% RSLogix 500 project TRAFFIC LIGHT.RSS, saved by version 8.30.00.16 %
PROJECT "UNTITLED"    % processor: MicroLogix 1000 %

PROGRAM FILES
  LAD 2 "MAIN_PROG"  11 rungs
  LAD 3 "FLASHER"  5 rungs
  LAD 4 "TIMER"  8 rungs
  LAD 5 "STI_INT"  1 rungs
  LAD 6, 7, 8, 9, 10, 11, 12, 13, 14, 15, 16: only END

DATA FILES
  O0 OUTPUT  1 elements
  I1 INPUT  2 elements
  S2 STATUS  33 elements
  B3 BINARY  32 elements
  T4 TIMER  40 elements
  C5 COUNTER  32 elements
  R6 CONTROL  16 elements
  N7 INTEGER  105 elements

LADDER 2 "MAIN_PROG"
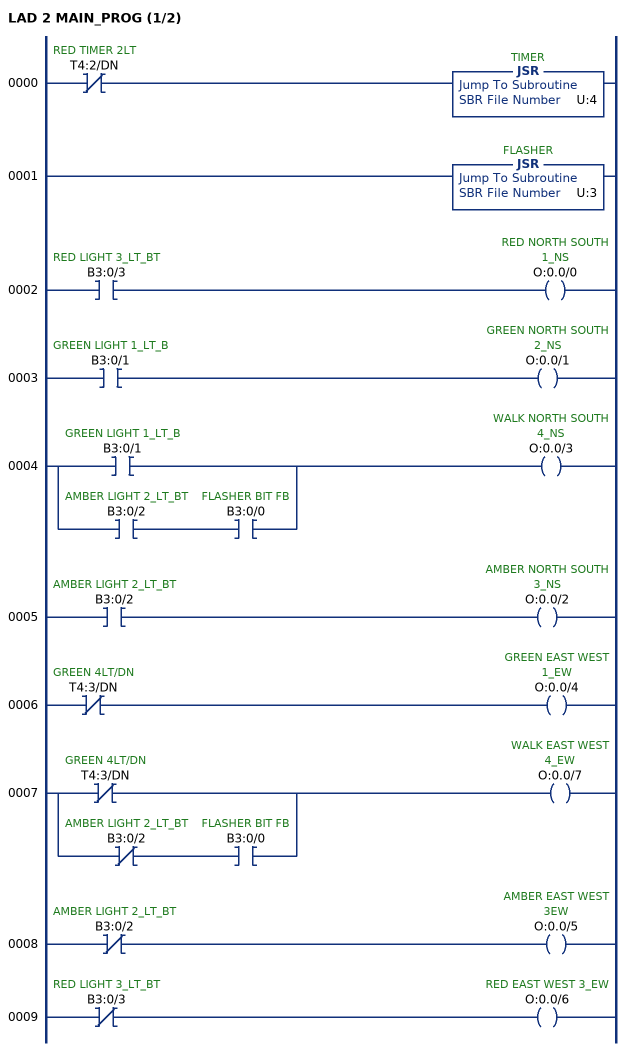
% Rung: 0 %
SOR XIO T4:2/DN JSR U:4 EOR
%   T4:2/DN  2LT  "RED TIMER" %
%   U:4  "TIMER" %
% Rung: 1 %
SOR JSR U:3 EOR
%   U:3  "FLASHER" %
% Rung: 2 %
SOR XIC B3:0/3 OTE O:0.0/0 EOR
%   B3:0/3  3_LT_BT  "RED LIGHT" %
%   O:0.0/0  1_NS  "RED NORTH SOUTH" %
% Rung: 3 %
SOR XIC B3:0/1 OTE O:0.0/1 EOR
%   B3:0/1  1_LT_B  "GREEN LIGHT" %
%   O:0.0/1  2_NS  "GREEN NORTH SOUTH" %
% Rung: 4 %
SOR BST XIC B3:0/1 NXB XIC B3:0/2 XIC B3:0/0 BND OTE O:0.0/3 EOR
%   B3:0/1  1_LT_B  "GREEN LIGHT" %
%   B3:0/2  2_LT_BT  "AMBER LIGHT" %
%   B3:0/0  FB  "FLASHER BIT" %
%   O:0.0/3  4_NS  "WALK NORTH SOUTH" %
% Rung: 5 %
SOR XIC B3:0/2 OTE O:0.0/2 EOR
%   B3:0/2  2_LT_BT  "AMBER LIGHT" %
%   O:0.0/2  3_NS  "AMBER NORTH SOUTH" %
% Rung: 6 %
SOR XIO T4:3/DN OTE O:0.0/4 EOR
%   T4:3  4LT  "GREEN" %
%   O:0.0/4  1_EW  "GREEN EAST WEST" %
% Rung: 7 %
SOR BST XIO T4:3/DN NXB XIO B3:0/2 XIC B3:0/0 BND OTE O:0.0/7 EOR
%   T4:3  4LT  "GREEN" %
%   B3:0/2  2_LT_BT  "AMBER LIGHT" %
%   B3:0/0  FB  "FLASHER BIT" %
%   O:0.0/7  4_EW  "WALK EAST WEST" %
% Rung: 8 %
SOR XIO B3:0/2 OTE O:0.0/5 EOR
%   B3:0/2  2_LT_BT  "AMBER LIGHT" %
%   O:0.0/5  3EW  "AMBER EAST WEST" %
% Rung: 9 %
SOR XIO B3:0/3 OTE O:0.0/6 EOR
%   B3:0/3  3_LT_BT  "RED LIGHT" %
%   O:0.0/6  3_EW  "RED EAST WEST" %

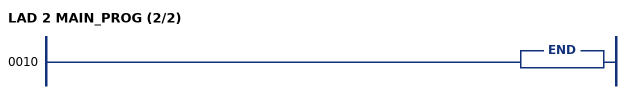
% Rung: 10 %
SOR END EOR

LADDER 3 "FLASHER"
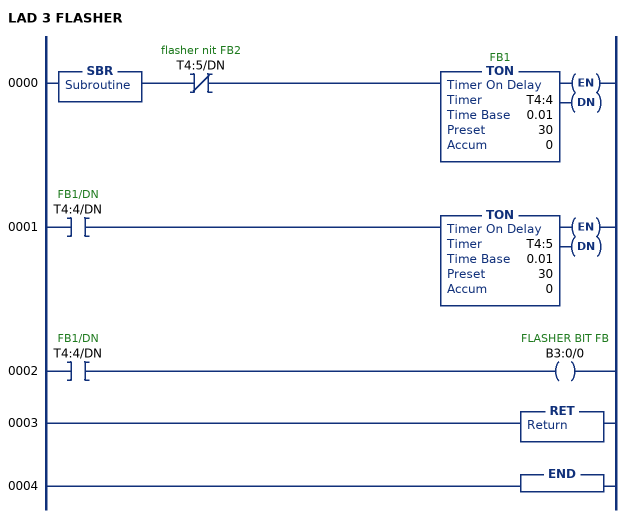
% Rung: 0 %
SOR SBR XIO T4:5/DN TON T4:4 0.01 30 0 EOR
%   T4:5/DN  FB2  "flasher nit" %
%   T4:4  FB1 %
% Rung: 1 %
SOR XIC T4:4/DN TON T4:5 0.01 30 0 EOR
%   T4:4  FB1 %
% Rung: 2 %
SOR XIC T4:4/DN OTE B3:0/0 EOR
%   T4:4  FB1 %
%   B3:0/0  FB  "FLASHER BIT" %
% Rung: 3 %
SOR RET EOR
% Rung: 4 %
SOR END EOR

LADDER 4 "TIMER"
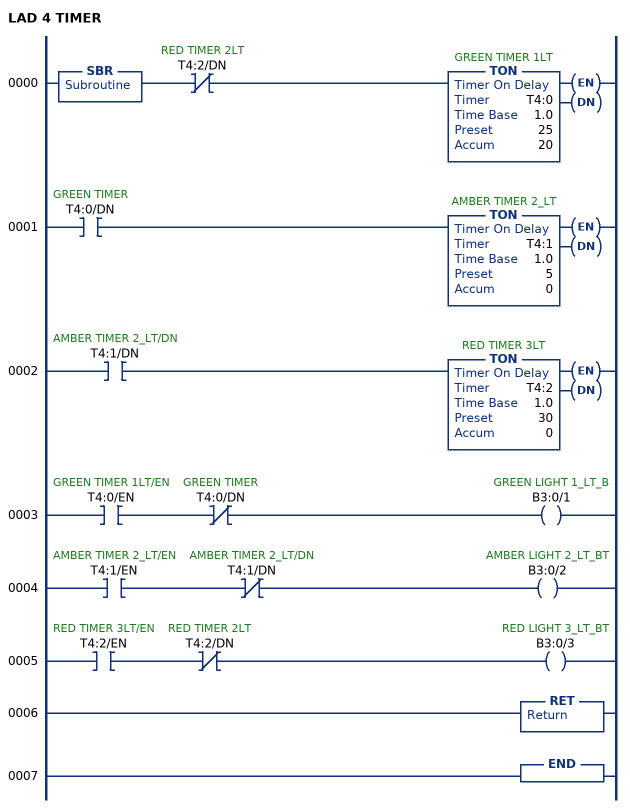
% Rung: 0 %
SOR SBR XIO T4:2/DN TON T4:0 1.0 25 20 EOR
%   T4:2/DN  2LT  "RED TIMER" %
%   T4:0  1LT  "GREEN TIMER" %
% Rung: 1 %
SOR XIC T4:0/DN TON T4:1 1.0 5 0 EOR
%   T4:0/DN  "GREEN TIMER" %
%   T4:1  2_LT  "AMBER TIMER" %
% Rung: 2 %
SOR XIC T4:1/DN TON T4:2 1.0 30 0 EOR
%   T4:1  2_LT  "AMBER TIMER" %
%   T4:2  3LT  "RED TIMER" %
% Rung: 3 %
SOR XIC T4:0/EN XIO T4:0/DN OTE B3:0/1 EOR
%   T4:0  1LT  "GREEN TIMER" %
%   T4:0/DN  "GREEN TIMER" %
%   B3:0/1  1_LT_B  "GREEN LIGHT" %
% Rung: 4 %
SOR XIC T4:1/EN XIO T4:1/DN OTE B3:0/2 EOR
%   T4:1  2_LT  "AMBER TIMER" %
%   B3:0/2  2_LT_BT  "AMBER LIGHT" %
% Rung: 5 %
SOR XIC T4:2/EN XIO T4:2/DN OTE B3:0/3 EOR
%   T4:2  3LT  "RED TIMER" %
%   T4:2/DN  2LT  "RED TIMER" %
%   B3:0/3  3_LT_BT  "RED LIGHT" %
% Rung: 6 %
SOR RET EOR
% Rung: 7 %
SOR END EOR

OTHER DOCUMENTED ADDRESSES
  O:0.0/8  "FLASHER BIT"
  U:5  "TIMER"

DATA TABLE (non-zero values as saved)
DATA T4
% .PRE .ACC %
% T4:0 % 25 20
% T4:1 % 5 0
% T4:2 % 30 0
% T4:3 % 25 0
% T4:4 % 30 0
% T4:5 % 30 0
